FUNCTION average : LREAL
VAR_IN_OUT
	aData : ARRAY[*] OF LREAL;
END_VAR
VAR
	nIdx  : DINT;
	fAmount, fSum : LREAL;
END_VAR

fAmount := 0;
FOR nIdx := LOWER_BOUND(aData,1) TO UPPER_BOUND(aData,1) DO
	fAmount := fAmount + 1;
    fSum := fSum + aData[nIdx] ;
END_FOR

average := fSum / fAmount;

END_FUNCTION

(* stored: Version 1.1.0.1, ProductVersion 3.1.4024.12
   POU average: Id {b4c02b53-6ff4-4574-acb6-cb645834b651}, SpecialFunc None *)
